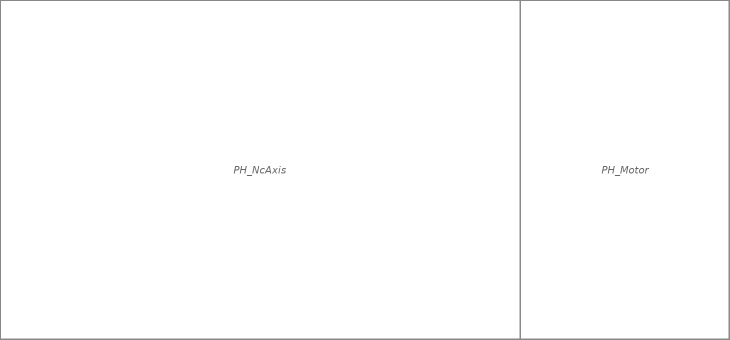
VISUALIZATION PH_AxisOnline_1  // 730x340
//==================================================================================================
//							Beckhoff Automation Poland
//									18.04.2018
//	Wizualizacja dla Axis Online
//  v1.0	|| TC v 3.1.4022.16		|| - pierwsza wersja
//==================================================================================================
VAR_IN_OUT
	stMcAxisOnline			: ST_McAxisOnline;	
END_VAR
    Frame (0,0 520x340)
        shows PH_NcAxis(stMcAxisOnline := stMcAxisOnline)
    Frame (520,0 210x340)
        shows PH_Motor(stMcAxisOnline := stMcAxisOnline)
END_VISUALIZATION

(* stored: Version 1.1.0.1, ProductVersion 3.1.4022.10
   Visu PH_AxisOnline_1: Id {62164ef7-fa3a-466a-beb5-98b957af37be} *)
